ABB RobotStudio station: MINIPROYECTO_MESA25.rspag

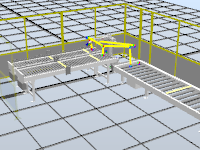
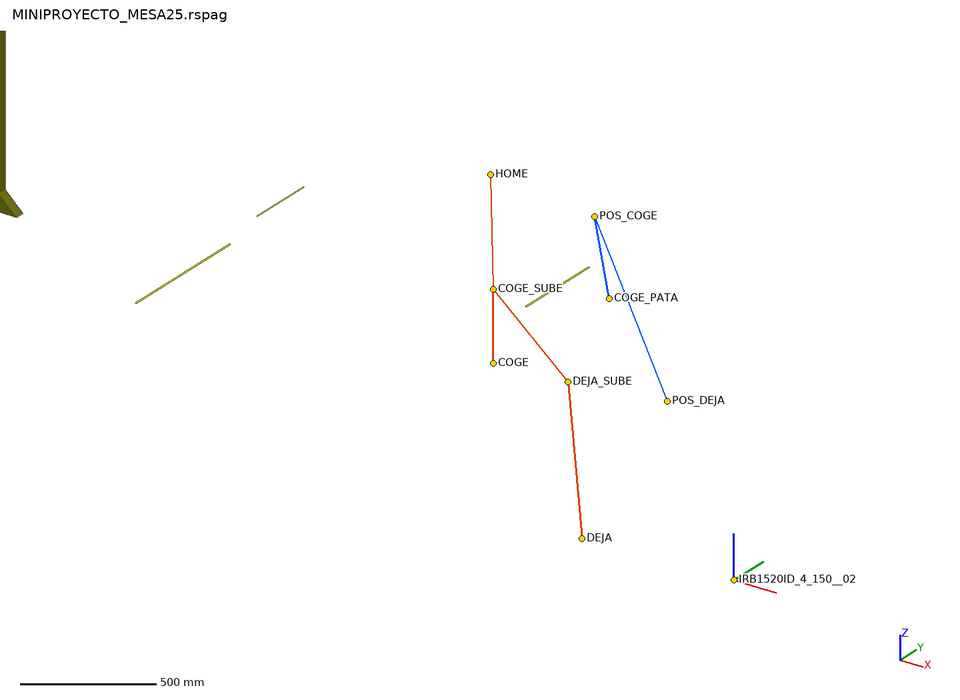
[picture v1: parts stored in the station drawn from their meshes, with robot base, taught points and paths (robot models come from the ABB library and are not in the file)]
--- station ---
Station MINIPROYECTO_MESA (saved by RobotStudio 21.2.9526.0)
Controller Controlador1, task T_ROB1: task frame (RAPID world) sits at (0, 0, 230) mm in the station
Controller Controlador1
  mechanical unit ROB_1: IRB1520ID_4_150__02, 6 joints, base frame (0, 0, -230) mm, rotated rx 0 ry 0 rz 180 deg
Layout (positions relative to the parent item):
  - CINTA_TABLERO [part, from Equipment\Conveyor Guide 600.rslib] at (-3500, -700, 0) mm
  - CINTA_PATAS [part, from Equipment\Conveyor Guide 400.rslib] at (-3500, 100, 0) mm
  - CINTA_CAJA_d [part, from Equipment\Conveyor 950 4000 h2.rslib] at (-400, -500, 0) mm, rotated rx 0 ry 0 rz -90 deg
  - IRB1520ID_4_150__02 [mechanism, from Robots\IRB1520ID_4_150_G_02.rslib] at (0, 0, 0) mm, rotated rx 0 ry 0 rz 180 deg; joint values [0, 0, 0, 0, 0.5236, 0] (rad or m)
  - CINTA_PATAS_SMC [part] at (-500, 500, 769) mm, rotated rx 0 ry 0 rz 180 deg, size 3000 x 400 x 5 mm
  - SC_CINTA_TABLERO [smart component]
      signals: DO PIEZA_OK, DI Activar_vacio, DI Desactivar_vacio, DI ACTIVAR_CINTA, DI MAS_PIEZA, DI MAS_PIEZA2
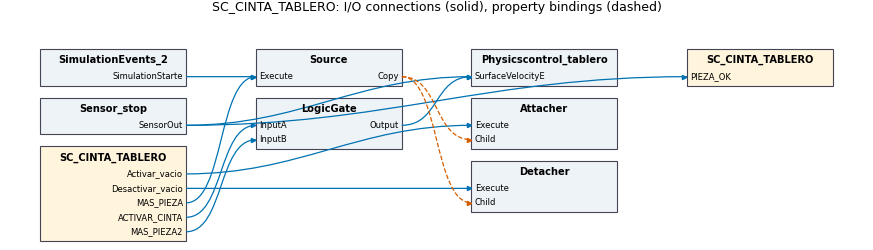
      connections:
        SimulationEvents_2.SimulationStarted -> Source.Execute
        Sensor_stop.SensorOut -> Physicscontrol_tablero.SurfaceVelocityEnabled
        Sensor_stop.SensorOut -> SC_CINTA_TABLERO.PIEZA_OK
        SC_CINTA_TABLERO.Activar_vacio -> Attacher.Execute
        SC_CINTA_TABLERO.Desactivar_vacio -> Detacher.Execute
        SC_CINTA_TABLERO.MAS_PIEZA -> Source.Execute
        SC_CINTA_TABLERO.ACTIVAR_CINTA -> LogicGate.InputA
        SC_CINTA_TABLERO.MAS_PIEZA2 -> LogicGate.InputB
        LogicGate.Output -> Physicscontrol_tablero.SurfaceVelocityEnabled
        Source.Copy => Attacher.Child
        Source.Copy => Detacher.Child
    - CINTA_TABLERO_SMC [part] at (-500, -100, 769) mm, rotated rx 0 ry 0 rz 180 deg, size 3000 x 600 x 5 mm
    - TABLERO [part] at (-3175, -405, 900) mm, size 550 x 550 x 50 mm
    - Source [smart component, from Components\Source.rslib]
        properties: Source=TABLERO; Copy=(none); Parent=(none); Position=[-3.175 -0.405 0.9]; Orientation=[0 0 0]; Transient=true; PhysicsBehavior=3
    - Sensor_+pieza [smart component, from Components\LineSensor.rslib]
        properties: Start=[-2.19 -0.7 0.8]; End=[-2.19 -0.1 0.8]; Radius=0.003; SensedPart=(none); SensedPoint=[0 0 0]
      - _sensorPart_ [part], size 6 x 600 x 6 mm
    - Sensor_stop [smart component, from Components\LineSensor.rslib]
        properties: Start=[-1.1 -0.1 0.8]; End=[-1.1 -0.69 0.8]; Radius=0; SensedPart=(none); SensedPoint=[0 0 0]
      - _sensorPart_ [part], size 0 x 590 x 0 mm
    - SimulationEvents_2 [smart component, from Components\SimulationEvents.rslib]
    - Attacher [smart component, from Components\Attacher.rslib]
        properties: Parent=PINZA_VACIO; Flange=0; Child=(none); Mount=false; Offset=[0 0 0]; Orientation=[0 0 0]
    - Detacher [smart component, from Components\Detacher.rslib]
        properties: Child=(none); KeepPosition=true
    - Physicscontrol_tablero [smart component, from Components\PhysicsControl.rslib]
        properties: Object=CINTA_TABLERO_SMC; Behavior=1; SurfaceVelocity=0.2
    - LogicGate [smart component, from Components\LogicGate.rslib]
        properties: Operator=AND; Delay=0
  - SC_CINTA_PATAS [smart component]
      signals: DI Activa_vacio, DI Desactiva_vacio, DO PIEZA_OK, DI ACTIVAR_CINTA, DI MAS_PIEZA, DI Activar_cinta
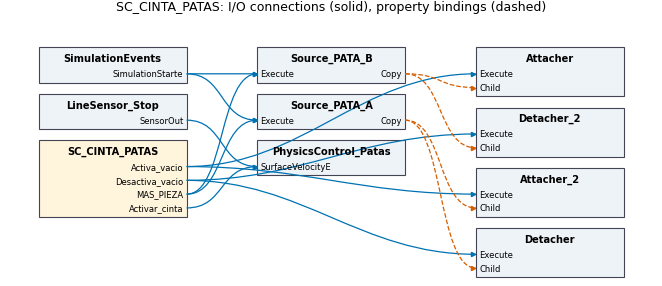
      connections:
        SimulationEvents.SimulationStarted -> Source_PATA_B.Execute
        SimulationEvents.SimulationStarted -> Source_PATA_A.Execute
        LineSensor_Stop.SensorOut -> PhysicsControl_Patas.SurfaceVelocityEnabled
        SC_CINTA_PATAS.Activa_vacio -> Attacher.Execute
        SC_CINTA_PATAS.Activa_vacio -> Attacher_2.Execute
        SC_CINTA_PATAS.Desactiva_vacio -> Detacher.Execute
        SC_CINTA_PATAS.Desactiva_vacio -> Detacher_2.Execute
        SC_CINTA_PATAS.MAS_PIEZA -> Source_PATA_B.Execute
        SC_CINTA_PATAS.MAS_PIEZA -> Source_PATA_A.Execute
        SC_CINTA_PATAS.Activar_cinta -> PhysicsControl_Patas.SurfaceVelocityEnabled
        Source_PATA_B.Copy => Attacher.Child
        Source_PATA_A.Copy => Attacher_2.Child
        Source_PATA_B.Copy => Detacher_2.Child
        Source_PATA_A.Copy => Detacher.Child
    - Source_PATA_A [smart component, from Components\Source.rslib] at (-500.83, 665.61, -264.15) mm, rotated rx 13.59 ry 9.71 rz 21.21 deg
        properties: Source=PATA_A; Copy=(none); Parent=(none); Position=[-3.175 0.265 0.9]; Orientation=[0 0 0]; Transient=true; PhysicsBehavior=3
    - LineSensor_+Pieza [smart component, from Components\LineSensor.rslib]
        properties: Start=[-2.243 0.15 0.8]; End=[-2.243 0.45 0.8]; Radius=0.002; SensedPart=(none); SensedPoint=[0 0 0]
      - _sensorPart_ [part], size 4 x 300 x 4 mm
    - PATA_A [part] at (-3175, 265, 900) mm, size 450 x 50 x 50 mm
    - PATA_B [part] at (-3175, 325, 900) mm, size 450 x 50 x 50 mm
    - Source_PATA_B [smart component, from Components\Source.rslib] at (-500.83, 665.61, -264.15) mm, rotated rx 13.59 ry 9.71 rz 21.21 deg
        properties: Source=PATA_B; Copy=(none); Parent=(none); Position=[-3.175 0.325 0.9]; Orientation=[0 0 0]; Transient=true; PhysicsBehavior=3
    - SimulationEvents [smart component, from Components\SimulationEvents.rslib]
    - PhysicsControl_Patas [smart component, from Components\PhysicsControl.rslib]
        properties: Object=CINTA_PATAS_SMC; Behavior=1; SurfaceVelocity=0.1
    - LineSensor_Stop [smart component, from Components\LineSensor.rslib]
        properties: Start=[-1 0.1 0.8]; End=[-1 0.5 0.8]; Radius=0.003; SensedPart=(none); SensedPoint=[0 0 0]
      - _sensorPart_ [part], size 6 x 400 x 6 mm
    - Attacher [smart component, from Components\Attacher.rslib]
        properties: Parent=PINZA_VACIO; Flange=0; Child=(none); Mount=false; Offset=[0 0 0]; Orientation=[0 0 0]
    - Attacher_2 [smart component, from Components\Attacher.rslib]
        properties: Parent=PINZA_VACIO; Flange=0; Child=(none); Mount=false; Offset=[0 0 0]; Orientation=[0 0 0]
    - Detacher [smart component, from Components\Detacher.rslib]
        properties: Child=Source_PATA_A; KeepPosition=true
    - Detacher_2 [smart component, from Components\Detacher.rslib]
        properties: Child=Source_PATA_B; KeepPosition=true
  - SC_CINTA_CAJA [smart component] at (-500, 500, 769) mm, rotated rx 0 ry 0 rz 180 deg
      signals: DI PARAR_CINTA_INICIO, DO CAJA_OK, DO MAS_TABLERO
      connections:
        SimulationEvents_3.SimulationStarted -> Source_3.Execute
        LineSensor_2.SensorOut -> Source_3.Execute
        SimulationEvents_3.SimulationStarted -> Source.Execute
        LineSensor_2.SensorOut -> Source.Execute
        LineSensor_2.SensorOut -> Physicscontrol_caja.SurfaceVelocityEnabled
        SC_CINTA_CAJA.PARAR_CINTA_INICIO -> Physicscontrol_caja.SurfaceVelocityEnabled
        Source.Executed -> SC_CINTA_CAJA.CAJA_OK
    - CINTA_CAJA_SMC [part] at (-100, 1000, -359) mm, rotated rx 0 ry 0 rz 90 deg, size 4000 x 910 x 5 mm
    - CAJA [part] at (-545, 1395, -169) mm, rotated rx 0 ry 0 rz 180 deg, size 856.3 x 654.8 x 107 mm
    - SimulationEvents_3 [smart component, from Components\SimulationEvents.rslib]
    - LineSensor_2 [smart component, from Components\LineSensor.rslib]
        properties: Start=[-0.1 3.454 -0.319]; End=[-1.01 3.454 -0.319]; Radius=0.002; SensedPart=(none); SensedPoint=[0 0 0]
      - _sensorPart_ [part], size 910 x 4 x 4 mm
    - Source [smart component, from Components\Source.rslib] at (3000, 400, -769) mm, rotated rx 0 ry 0 rz 180 deg
        properties: Source=CAJA; Copy=(none); Parent=(none); Position=[-0.545 1.4 -0.2]; Orientation=[0 0 0]; Transient=true; PhysicsBehavior=3
  - PINZA_VACIO [mechanism, from Libraries\PINZA_VACIO.rslib] at (-1056.21, 0, 1143) mm, rotated rx 180 ry 60 rz 0 deg
  - VALLA1 [graphiccomponentgroup, from Equipment\Fence_2500.rslib] at (1000, 1000, 0) mm, rotated rx 0 ry 0 rz 90 deg
    - Body 1 [part, from Equipment\Fence_2500.rslib]
    - Body 2 [part, from Equipment\Fence_2500.rslib]
  - PUERTA [graphiccomponentgroup, from Equipment\Fence_Gate.rslib] at (1000, -500, 0) mm
    - Body 1 [part, from Equipment\Fence_Gate.rslib]
    - Body 2 [part, from Equipment\Fence_Gate.rslib]
    - Body 3 [part, from Equipment\Fence_Gate.rslib]
  - Valla2 [graphiccomponentgroup, from Equipment\Fence_2500.rslib] at (1000, -3000, 0) mm
    - Body 1 [part, from Equipment\Fence_2500.rslib]
    - Body 2 [part, from Equipment\Fence_2500.rslib]
  - Valla3 [graphiccomponentgroup, from Equipment\Fence_2500.rslib] at (1000, -5500, 0) mm
    - Body 1 [part, from Equipment\Fence_2500.rslib]
    - Body 2 [part, from Equipment\Fence_2500.rslib]
  - VALLA4 [graphiccomponentgroup, from Equipment\Fence_2500.rslib] at (-1500, 1000, 0) mm, rotated rx 0 ry 0 rz 90 deg
    - Body 1 [part, from Equipment\Fence_2500.rslib]
    - Body 2 [part, from Equipment\Fence_2500.rslib]
  - VALLA5 [graphiccomponentgroup] at (-4000, 1000, 0) mm, rotated rx 0 ry 0 rz 180 deg
    - Body 1 [part], size 200 x 2500 x 2000 mm
    - Body 2 [part], size 5 x 2420 x 710 mm
  - Physicscontrol_caja [smart component, from Components\PhysicsControl.rslib] at (-500, 500, 769) mm, rotated rx 0 ry 0 rz 180 deg
      properties: Object=CINTA_CAJA_SMC; Behavior=1; SurfaceVelocity=0.2
Attachment: SC_CINTA_CAJA is attached to CINTA_PATAS_SMC
Attachment: Source is attached to CINTA_PATAS
Attachment: PINZA_VACIO is attached to IRB1520ID_4_150__02 / Link6
Attachment: WorkTablero is attached to CINTA_TABLERO_SMC
Attachment: Source_PATA_A is attached to PINZA_VACIO / PINZA_VACIO
Attachment: Source_PATA_B is attached to PINZA_VACIO / PINZA_VACIO
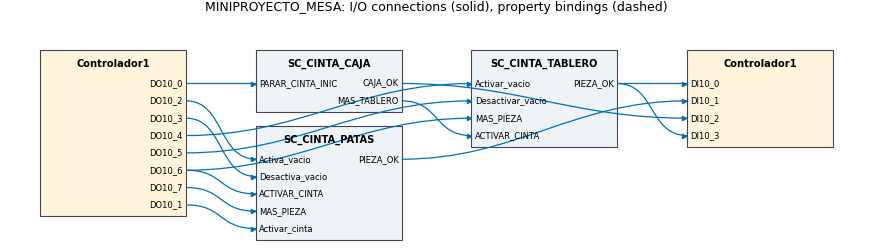
Station logic (signal -> signal, property => property):
  Controlador1.DO10_0 -> SC_CINTA_CAJA.PARAR_CINTA_INICIO
  Controlador1.DO10_2 -> SC_CINTA_PATAS.Activa_vacio
  Controlador1.DO10_3 -> SC_CINTA_PATAS.Desactiva_vacio
  SC_CINTA_TABLERO.PIEZA_OK -> Controlador1.DI10_0
  SC_CINTA_PATAS.PIEZA_OK -> Controlador1.DI10_1
  SC_CINTA_CAJA.CAJA_OK -> Controlador1.DI10_2
  SC_CINTA_TABLERO.PIEZA_OK -> Controlador1.DI10_3
  Controlador1.DO10_4 -> SC_CINTA_TABLERO.Activar_vacio
  Controlador1.DO10_5 -> SC_CINTA_TABLERO.Desactivar_vacio
  Controlador1.DO10_6 -> SC_CINTA_PATAS.ACTIVAR_CINTA
  Controlador1.DO10_7 -> SC_CINTA_PATAS.MAS_PIEZA
  Controlador1.DO10_1 -> SC_CINTA_PATAS.Activar_cinta
  Controlador1.DO10_6 -> SC_CINTA_TABLERO.MAS_PIEZA
  SC_CINTA_CAJA.MAS_TABLERO -> SC_CINTA_TABLERO.ACTIVAR_CINTA

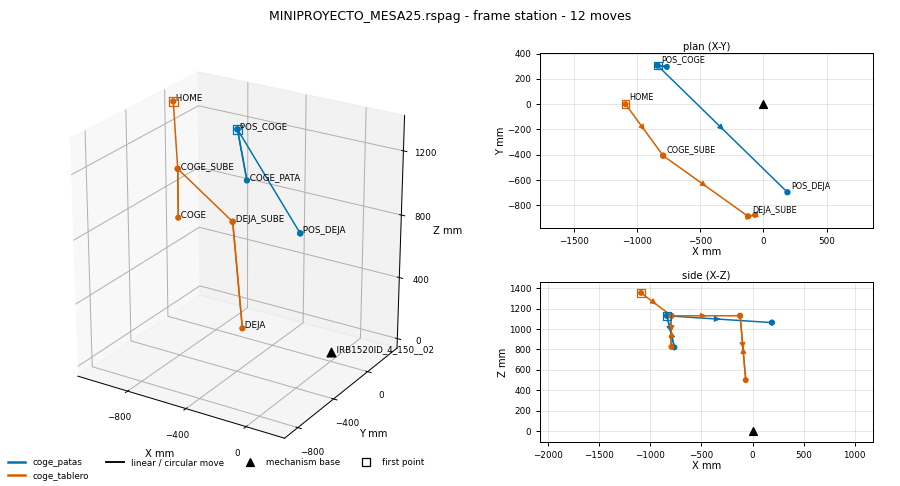
[picture p0: tool path of MINIPROYECTO_MESA25.rspag in frame station, 12 of 13 moves have a stored position in this frame; points joined in program order, loops and branches not executed]
--- Backups/Controlador1/RAPID/TASK1/PROGMOD/CalibData.mod ---
MODULE CalibData
    PERS tooldata PINZA_VACIO:=[TRUE,[[0,0,40],[1,0,0,0]],[2,[0,0,1],[1,0,0,0],0,0,0]];
    TASK PERS wobjdata WorkTablero:=[FALSE,TRUE,"",[[-500,-100,539],[0,0,0,1]],[[0,0,0],[1,0,0,0]]];
    TASK PERS wobjdata WorkPatas:=[FALSE,TRUE,"",[[0,0,0],[1,0,0,0]],[[0,0,0],[1,0,0,0]]];
ENDMODULE

--- Backups/Controlador1/RAPID/TASK1/PROGMOD/Module1.mod ---
MODULE Module1
        CONST robtarget HOME:=[[-1090.846096908,0,1123],[0,0.866025404,0,-0.5],[0,0,0,0],[9E+09,9E+09,9E+09,9E+09,9E+09,9E+09]];
    CONST robtarget COGE_SUBE:=[[293.363530459,307.256897821,360.384099828],[0.013096782,0.679377704,0.733666808,0.002724996],[0,-1,1,0],[9E+09,9E+09,9E+09,9E+09,9E+09,9E+09]];
    CONST robtarget POS_A_COGER:=[[293.363483733,307.256806105,84.836573661],[0.01309679,0.679377678,0.733666832,0.00272501],[-2,-1,1,0],[9E+09,9E+09,9E+09,9E+09,9E+09,9E+09]];
    CONST robtarget POS_A_DEJAR:=[[-379.121119695,783.111493971,470.871022461],[0.013096759,0.679377706,0.733666806,0.002725024],[-2,-1,1,0],[9E+09,9E+09,9E+09,9E+09,9E+09,9E+09]];
    CONST robtarget DEJA:=[[-433.608396871,775.808738791,-269.012556748],[0.009904467,-0.040327135,0.999113273,0.006949172],[0,-1,0,0],[9E+09,9E+09,9E+09,9E+09,9E+09,9E+09]];
    CONST robtarget POS_A_DEJAR_2:=[[-379.121119695,783.111493971,470.871022461],[0.013096759,0.679377706,0.733666806,0.002725024],[-2,-1,1,0],[9E+09,9E+09,9E+09,9E+09,9E+09,9E+09]];
    CONST robtarget COGE:=[[293.36353877,307.256902247,56.879691539],[0.013096779,0.679377717,0.733666795,0.002724989],[-2,-1,1,0],[9E+09,9E+09,9E+09,9E+09,9E+09,9E+09]];
    CONST robtarget Target_10:=[[-837.743841333,305.727222369,899.384048226],[0.00202243,0.052965018,-0.998506763,-0.013223498],[-1,-1,1,0],[9E+09,9E+09,9E+09,9E+09,9E+09,9E+09]];
    CONST robtarget Target_20:=[[-392.489923305,691.64804172,-289.463687721],[0.009719164,-0.014159579,0.999826543,0.007206059],[0,-1,0,0],[9E+09,9E+09,9E+09,9E+09,9E+09,9E+09]];
    CONST robtarget DEJA_SUBE:=[[-378.672044822,787.098067668,360.460176589],[0.01321686,-0.00460022,0.999820673,0.012758284],[0,-1,0,0],[9E+09,9E+09,9E+09,9E+09,9E+09,9E+09]];
    CONST robtarget Target_30:=[[-804.22598647,294.236504471,564.95990756],[0.000500133,-0.018236855,0.999761158,0.012033063],[-1,-1,1,0],[9E+09,9E+09,9E+09,9E+09,9E+09,9E+09]];
    CONST robtarget Target_40:=[[189.644354203,-696.850059522,832.736095493],[0.029410487,0.698598159,-0.714296574,0.029597962],[1,-1,2,0],[9E+09,9E+09,9E+09,9E+09,9E+09,9E+09]];
    CONST robtarget Target_50:=[[183.853159454,-865.181419069,199.977231946],[0.004842738,0.698770008,-0.715215791,-0.012782668],[1,-1,2,0],[9E+09,9E+09,9E+09,9E+09,9E+09,9E+09]];
!***********************************************************
    !
    ! Módulo:  Module1
    !
    ! Descripción:
    !   <Introduzca la descripción aquí>
    !
    ! Autor: estev
    !
    ! Versión: 1.0
    !
    !***********************************************************


    !***********************************************************
    !
    ! Procedimiento Main
    !
    !   Este es el punto de entrada de su programa
    !
    !***********************************************************
    VAR num ciclo:=0;
    CONST robtarget POS_COGE:=[[-837.743841333,305.727222369,899.384048226],[0.00202243,0.052965018,-0.998506763,-0.013223498],[-1,-1,1,0],[9E+09,9E+09,9E+09,9E+09,9E+09,9E+09]];
    CONST robtarget COGE_PATA:=[[-764.266641527,295.09265747,590.010212024],[0.000500133,-0.018236855,0.999761158,0.012033063],[-1,-1,1,0],[9E+09,9E+09,9E+09,9E+09,9E+09,9E+09]];
    CONST robtarget POS_DEJA:=[[189.644354203,-696.850059522,832.736095493],[0.029410487,0.698598159,-0.714296574,0.029597962],[1,-1,2,0],[9E+09,9E+09,9E+09,9E+09,9E+09,9E+09]];
    CONST robtarget DEJA_PATA:=[[271.823306057,-847.304219732,273.497727896],[0.001857985,-0.717262768,0.696765796,0.006935133],[1,-1,2,0],[9E+09,9E+09,9E+09,9E+09,9E+09,9E+09]];
    VAR num despl;
    PROC main()
        Reset DO10_0;
        Reset DO10_6;
        Reset DO10_4;
        Reset DO10_2;
        Reset DO10_7;
        Reset DO10_1;
        IF DI10_0=1 ciclo:=1;
        IF ciclo=1 THEN
            coge_tablero;
            coge_patas;
            Waittime 3;
            Set DO10_7;
            Set DO10_1;
            Waittime 10;
            coge_patas;
            Reset DO10_7;
            Waittime 2;
            despl:=0;
            Set DO10_6;
            Set DO10_0;
            Waittime 9;
        ENDIF


    ENDPROC

    PROC coge_patas()

        MoveL POS_COGE,v200,z100,PINZA_VACIO\WObj:=WorkPatas;
        Waittime 10;
        MoveL COGE_PATA,v200,z100,PINZA_VACIO\WObj:=WorkPatas;
        Waittime 3;
        Set DO10_2;
        WaitTime 3;
        MoveL POS_COGE,v200,z100,PINZA_VACIO\WObj:=WorkPatas;
        MoveL POS_DEJA,v200,z100,PINZA_VACIO\WObj:=WorkPatas;
        Waittime 1;
        MoveL Offs (DEJA_PATA,0,0,despl),v200,z100,PINZA_VACIO\WObj:=WorkPatas;
        waittime 3;
        Reset DO10_2;
        Set DO10_3;
        MoveL POS_DEJA,v200,z100,PINZA_VACIO\WObj:=WorkPatas;
        Reset DO10_3;
        despl:= despl+50;
    ENDPROC
    PROC coge_tablero()
        MoveL HOME,v200,z100,PINZA_VACIO\WObj:=wobj0;
        MoveL COGE_SUBE,v200,z100,PINZA_VACIO\WObj:=WorkTablero;
        Waittime 15;
         MoveL COGE,v200,z100,PINZA_VACIO\WObj:=WorkTablero;
         WaitTime 3;
        Set DO10_4;
        WaitTime 3;
        MoveL COGE_SUBE,v200,z100,PINZA_VACIO\WObj:=WorkTablero;
        MoveL DEJA_SUBE,v200,z100,PINZA_VACIO\WObj:=WorkTablero;
        MoveL DEJA,v200,z100,PINZA_VACIO\WObj:=WorkTablero;
        Waittime 3;
        Reset DO10_4;
        Set DO10_5;
        MoveL DEJA_SUBE,v200,z100,PINZA_VACIO\WObj:=WorkTablero;
        Reset DO10_5;
    ENDPROC
ENDMODULE

--- Backups/Controlador1/SYSPAR/EIO.cfg ---
EIO:CFG_1.0:6:1::
#
INDUSTRIAL_NETWORK:

      -Name "DeviceNet" -Label "DeviceNet Master/Slave Network" -Address "2"
#
DEVICENET_DEVICE:

      -Name "d652" -VendorName "ABB Robotics" -ProductName "24 VDC I/O Device"\
      -Label "DSQC 652 24 VDC I/O Device" -Address 10 -ProductCode 26\
      -DeviceType 7 -ConnectionType "COS" -OutputSize 2 -InputSize 2
#
DEVICENET_INTERNAL_DEVICE:

      -Name "DN_Internal_Device" -VendorName "ABB Robotics"\
      -ProductName "DeviceNet Internal Slave Device"
#
EIO_SIGNAL:

      -Name "DO10_0" -SignalType "DO" -Device "d652" -DeviceMap "0"

      -Name "DO10_1" -SignalType "DO" -Device "d652" -DeviceMap "1"

      -Name "DO10_2" -SignalType "DO" -Device "d652" -DeviceMap "2"

      -Name "DO10_3" -SignalType "DO" -Device "d652" -DeviceMap "3"

      -Name "DO10_4" -SignalType "DO" -Device "d652" -DeviceMap "4"

      -Name "DO10_5" -SignalType "DO" -Device "d652" -DeviceMap "5"

      -Name "DO10_6" -SignalType "DO" -Device "d652" -DeviceMap "6"

      -Name "DO10_7" -SignalType "DO" -Device "d652" -DeviceMap "7"

      -Name "DI10_0" -SignalType "DI" -Device "d652" -DeviceMap "0"

      -Name "DI10_1" -SignalType "DI" -Device "d652" -DeviceMap "1"

      -Name "DI10_2" -SignalType "DI" -Device "d652" -DeviceMap "2"

      -Name "DI10_3" -SignalType "DI" -Device "d652" -DeviceMap "3"

      -Name "DI10_4" -SignalType "DI" -Device "d652" -DeviceMap "4"

      -Name "DI10_5" -SignalType "DI" -Device "d652" -DeviceMap "5"

      -Name "DI10_6" -SignalType "DI" -Device "d652" -DeviceMap "6"

      -Name "DI10_7" -SignalType "DI" -Device "d652" -DeviceMap "7"
